// TIA Portal V20 export
DATA_BLOCK "DB_DataFinalPart"   // DB700
{ S7_Optimized_Access := 'TRUE' }
// stored: AutoNumber false, MemoryReserve 100
   VAR
      FinalPart : Array[0..100] of "UDT_Tracability";
   END_VAR
BEGIN
END_DATA_BLOCK
